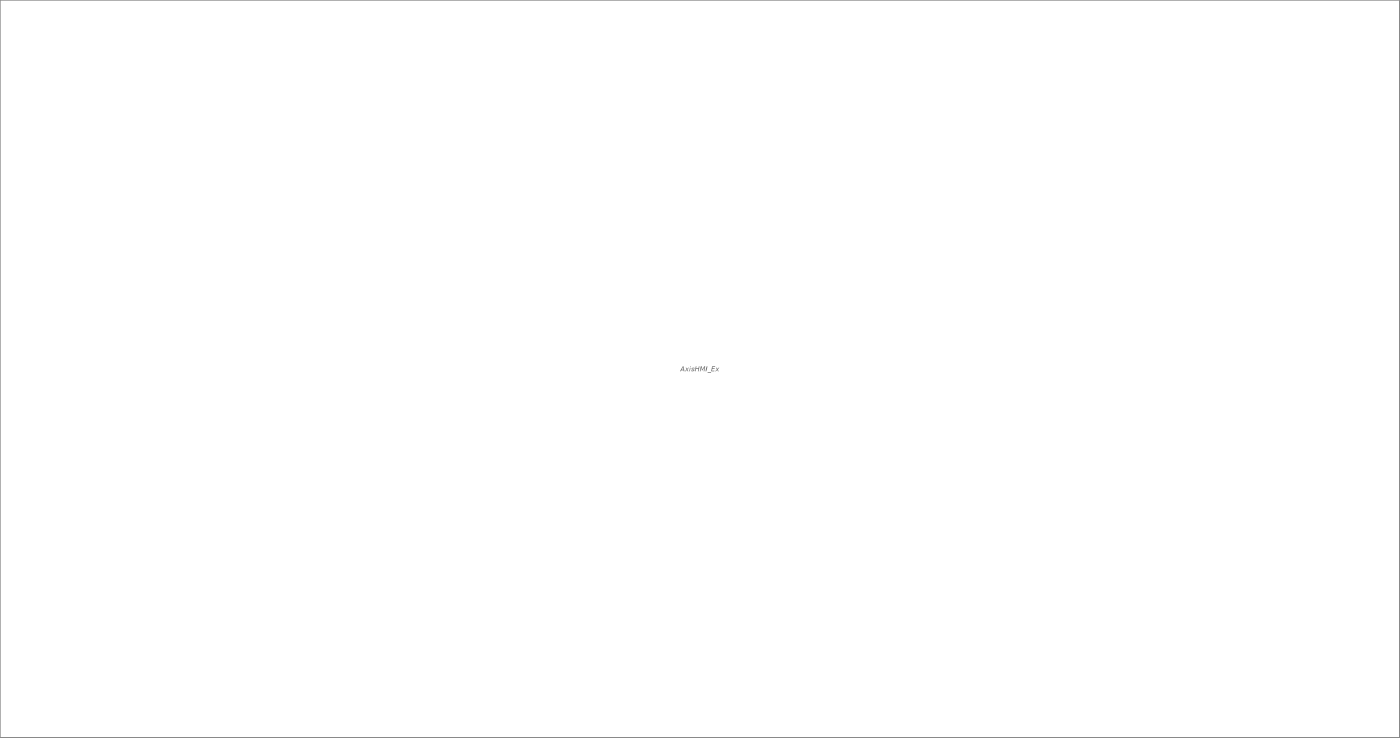
VISUALIZATION visu_autoStore  // 2048x1080
VAR_IN_OUT
	autoStore	: FB_autoStore;
END_VAR
    TabControl (0,0 2048x1080)
        shows AxisHMI_Ex(stAxisHMI := autoStore.st_mcAxis_lift, mcAxis := autoStore.mcAxis_lift, xError := autoStore.mcAxis_lift.xError)
        shows AxisHMI_Ex(stAxisHMI := autoStore.st_mcAxis_transfer, mcAxis := autoStore.mcAxis_transfer, xError := autoStore.mcAxis_transfer.xError)
        shows v_io_autoStore(autoStore := autoStore)
        shows AxisHMI_Ex(stAxisHMI := GVL.fb_working.st_mcAxis_vacuun[0], mcAxis := GVL.fb_working.mcAxis_vacuun[0], xError := GVL.fb_working.mcAxis_vacuun[0].xError)
        shows AxisHMI_Ex(stAxisHMI := GVL.fb_working.st_mcAxis_vacuun[1], mcAxis := GVL.fb_working.mcAxis_vacuun[1], xError := GVL.fb_working.mcAxis_vacuun[1].xError)
        shows AxisHMI_Ex(stAxisHMI := GVL.fb_working.st_mcAxis_bagOpen[0], mcAxis := GVL.fb_working.mcAxis_bagOpen[0], xError := GVL.fb_working.mcAxis_bagOpen[0].xError)
        shows AxisHMI_Ex(stAxisHMI := GVL.fb_working.st_mcAxis_bagOpen[1], mcAxis := GVL.fb_working.mcAxis_bagOpen[1], xError := GVL.fb_working.mcAxis_bagOpen[1].xError)
        shows AxisHMI_Ex(stAxisHMI := GVL.fb_working.st_mcAxis_bagOpen[2], mcAxis := GVL.fb_working.mcAxis_bagOpen[2], xError := GVL.fb_working.mcAxis_bagOpen[2].xError)
        shows AxisHMI_Ex(stAxisHMI := GVL.fb_working.st_mcAxis_bagOpen[3], mcAxis := GVL.fb_working.mcAxis_bagOpen[3], xError := GVL.fb_working.mcAxis_bagOpen[3].xError)
        [0]: TabTitle=Lift
        [1]: TabTitle=BagOpen
        [3]: TabTitle=Axis_vacuun_0
        [4]: TabTitle=Axis_vacuun_1
        [5]: TabTitle=Axis_bagOpen_0
        [6]: TabTitle=Axis_bagOpen_1
        [7]: TabTitle=Axis_bagOpen_2
        [8]: TabTitle=Axis_bagOpen_3
        p2837713833: gantrybase.mcAxis[EN_Axis.Z].sAxisName
END_VISUALIZATION

(* stored: Version 1.1.0.1, ProductVersion 3.1.4024.12
   Visu visu_autoStore: Id {39055b5a-8566-414b-ab66-0ec8df8099fa} *)
